// TIA Portal project "Project3" (V15.1)

(* hardware
DEVICE "S7300/ET200M station_1"  S7-300 station
   slot 0: "Rail_0"  Rail  6ES7 390-1***0-0AA0
   slot 2: "PLC_1"  CPU 312  6ES7 312-1AE13-0AB0  V2.6
      slot 0: "MPI interface_1"  X1
*)

// ===== PLC "PLC_1"  CPU 312 =====

VAR_GLOBAL   // PLC tag table "Default tag table"
   "LSL" AT %I0.0 : Bool;   // Level Switch Low (0 - nizak nivo)
   "LSH" AT %I0.1 : Bool;   // Level Switch High (0 - visok nivo)
   "LS" AT %I0.2 : Bool;   // Radni nivo (1 - dostignut nivo)
   "R/A" AT %I0.3 : Bool;   // 0 - Rucno, 1 - automatsko
   "Uklj_pumpe" AT %Q4.0 : Bool;   // Ukljucenje pumpe
   "Signalna lampica" AT %Q4.1 : Bool;   // Signalizacija rada
   "Rucni rezim rada" AT %M0.0 : Bool;
   "Rucni rezim rada SR" AT %M1.0 : Bool;
   "Automatski rezim rada" AT %M0.1 : Bool;
   "Automatski rezim rada SR" AT %M1.1 : Bool;
END_VAR

DATA_BLOCK "Data_block_1"   // DB20
{ S7_Optimized_Access := 'FALSE' }
VERSION : 0.1
   VAR
      Start_pumpe : Bool;
      Stop_pumpe : Bool;
   END_VAR
BEGIN
END_DATA_BLOCK

FUNCTION "Mode" : Void   // FC1, LAD
{ S7_Optimized_Access := 'FALSE' }
VERSION : 0.1
BEGIN

REGION Network 1: Ukljucenje pumpe
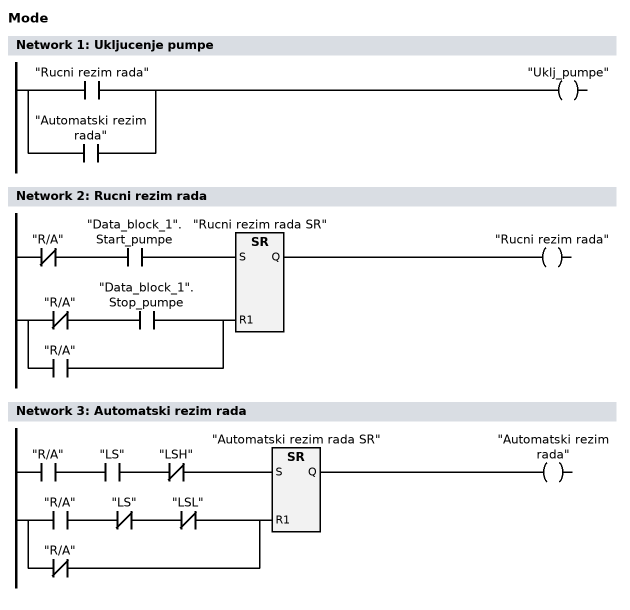
   RUNG wire#powerrail
      Contact( "Rucni rezim rada" )
      wire#w1
      Coil( "Uklj_pumpe" )
   END_RUNG
   RUNG wire#powerrail
      Contact( "Automatski rezim rada" )
   END_RUNG wire#w1
   // the same network as SCL:
   "Uklj_pumpe" := "Rucni rezim rada" OR "Automatski rezim rada";
END_REGION

REGION Network 2: Rucni rezim rada
   RUNG wire#powerrail
      I_Contact( "R/A" )
      Contact( "Data_block_1".Start_pumpe )
      S_SR(operand := "Rucni rezim rada SR", r1 := wire#w1)
      Coil( "Rucni rezim rada" )
   END_RUNG
   RUNG wire#powerrail
      I_Contact( "R/A" )
      Contact( "Data_block_1".Stop_pumpe )
   END_RUNG wire#w1
   RUNG wire#powerrail
      Contact( "R/A" )
   END_RUNG wire#w1
   // the same network as SCL:
   IF NOT "R/A" AND "Data_block_1".Start_pumpe THEN
       "Rucni rezim rada SR" := TRUE;   // SR flip-flop
   END_IF;
   IF (NOT "R/A" AND "Data_block_1".Stop_pumpe) OR "R/A" THEN "Rucni rezim rada SR" := FALSE; END_IF;
   "Rucni rezim rada" := "Rucni rezim rada SR";
END_REGION

REGION Network 3: Automatski rezim rada
   RUNG wire#powerrail
      Contact( "R/A" )
      Contact( "LS" )
      I_Contact( "LSH" )
      S_SR(operand := "Automatski rezim rada SR", r1 := wire#w1)
      Coil( "Automatski rezim rada" )
   END_RUNG
   RUNG wire#powerrail
      Contact( "R/A" )
      I_Contact( "LS" )
      I_Contact( "LSL" )
   END_RUNG wire#w1
   RUNG wire#powerrail
      I_Contact( "R/A" )
   END_RUNG wire#w1
   // the same network as SCL:
   IF "R/A" AND "LS" AND NOT "LSH" THEN
       "Automatski rezim rada SR" := TRUE;   // SR flip-flop
   END_IF;
   IF ("R/A" AND NOT "LS" AND NOT "LSL") OR NOT "R/A" THEN "Automatski rezim rada SR" := FALSE; END_IF;
   "Automatski rezim rada" := "Automatski rezim rada SR";
END_REGION
END_FUNCTION

ORGANIZATION_BLOCK "Main"   // OB1, LAD
TITLE = "Main Program Sweep (Cycle)"
{ S7_Optimized_Access := 'FALSE' }
VERSION : 0.1
   VAR_TEMP
      OB1_EV_CLASS : Byte;   // Bits 0-3 = 1 (Coming event), Bits 4-7 = 1 (Event class 1)
      OB1_SCAN_1 : Byte;   // 1 (Cold restart scan 1 of OB 1), 3 (Scan 2-n of OB 1)
      OB1_PRIORITY : Byte;   // Priority of OB Execution
      OB1_OB_NUMBR : Byte;   // 1 (Organization block 1, OB1)
      OB1_RESERVED_1 : Byte;   // Reserved for system
      OB1_RESERVED_2 : Byte;   // Reserved for system
      OB1_PREV_CYCLE : Int;   // Cycle time of previous OB1 scan (milliseconds)
      OB1_MIN_CYCLE : Int;   // Minimum cycle time of OB1 (milliseconds)
      OB1_MAX_CYCLE : Int;   // Maximum cycle time of OB1 (milliseconds)
      OB1_DATE_TIME : Date_And_Time;   // Date and time OB1 started
   END_VAR
BEGIN
END_ORGANIZATION_BLOCK